// TIA Portal V20 export
// export: Created 2026-04-11T06:02:30.6226391Z, ExportSetting WithDefaults, DisplayName Totally Integrated Automation Portal, DisplayVersion V20, DisplayName TIA Portal Openness, DisplayVersion V20, DisplayName TIA Portal Version Control Interface, DisplayVersion V20, DisplayName STEP 7 Professional, DisplayVersion V20, DisplayName STEP 7 Safety, DisplayVersion V20, DisplayName WinCC Basic/Comfort/Advanced, DisplayVersion V20, DisplayName WinCC Unified, DisplayVersion V20
TYPE "udtHMI_Brabender_Input"
// stored: IsFailsafeCompliant false
   STRUCT
      Status { ExternalWritable := 'False'} : "udtHMI_Brabender_Status";
      iAlarm { ExternalWritable := 'False'} : Int;   // Controller alarm number
      iStartConditionStatus { ExternalWritable := 'False'} : Int;   // Start conditions byte
      iOperatingMode { ExternalWritable := 'False'} : Int;   // Operating modes byte
      rDecadeSwitch { ExternalWritable := 'False'} : Real;   // Decade switch
      rActualSetpoint { ExternalWritable := 'False'} : Real;   // Actual Setpoint [kg/h]
      rActualFlow { ExternalWritable := 'False'} : Real;   // Actual Flow [kg/h]
      rActualWeight { ExternalWritable := 'False'} : Real;   // Actual Weight [kg]
      rActualSpeed { ExternalWritable := 'False'} : Real;   // Actual Speed [%]
      rActualThroughput { ExternalWritable := 'False'} : Real;   // Actual Throughput/Totalizer [kg]
      rActualSPAnalog { ExternalWritable := 'False'} : Real;   // Setpoint [%] for analogue control
      rActualSPCleaning { ExternalWritable := 'False'} : Real;   // Setpoint [%] for DI/cleaning
      rSamplingQuantity { ExternalWritable := 'False'} : Real;   // Sampling quantity [kg/h]
      rAutoTareValue { ExternalWritable := 'False'} : Real;   // Auto-tare value [kg]
      rControlDifference { ExternalWritable := 'False'} : Real;   // Control difference [%]
      rActualBulkDensity { ExternalWritable := 'False'} : Real;   // Bulk density [kg/l]
      rCheckMaxOutput { ExternalWritable := 'False'} : Real;   // Check. max. output [kg/hr]
      rActualPTermController { ExternalWritable := 'False'} : Real;   // P-term controller
      rActualITermController { ExternalWritable := 'False'} : Real;   // I-term controller
      rActualDTermController { ExternalWritable := 'False'} : Real;   // D-term controller
      rControllerAdaptation { ExternalWritable := 'False'} : Real;   // Controller adaptation
      rActualFillLevelMin { ExternalWritable := 'False'} : Real;   // Filling level minimum [%]
      rActualFillLevelMax { ExternalWritable := 'False'} : Real;   // Filling level maximum [%]
   END_STRUCT;
END_TYPE
